// Mitsubishi GX Works2 project: msp_7   PLC: Q03UDV

PROGRAM MAIN
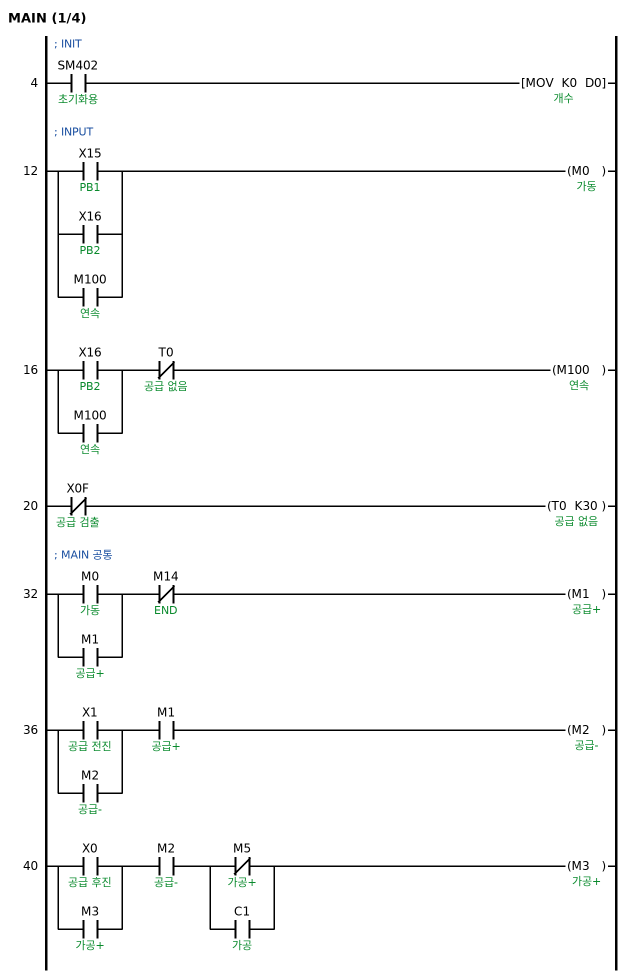
; INIT
4     LD      SM402  ; 초기화용
      MOV     K0 D0  ; 개수
; INPUT
12    LD      X15  ; PB1
      OR      X16  ; PB2
      OR      M100  ; 연속
      OUT     M0  ; 가동
16    LD      X16  ; PB2
      OR      M100  ; 연속
      ANI     T0  ; 공급 없음
      OUT     M100  ; 연속
20    LDI     X0F  ; 공급 검출
      OUT     T0 K30  ; 공급 없음
; MAIN 공통
32    LD      M0  ; 가동
      OR      M1  ; 공급+
      ANI     M14  ; END
      OUT     M1  ; 공급+
36    LD      X1  ; 공급 전진
      OR      M2  ; 공급-
      AND     M1  ; 공급+
      OUT     M2  ; 공급-
40    LD      X0  ; 공급 후진
      OR      M3  ; 가공+
      AND     M2  ; 공급-
      LDI     M5  ; 가공+
      OR      C1  ; 가공
      ANB
      OUT     M3  ; 가공+
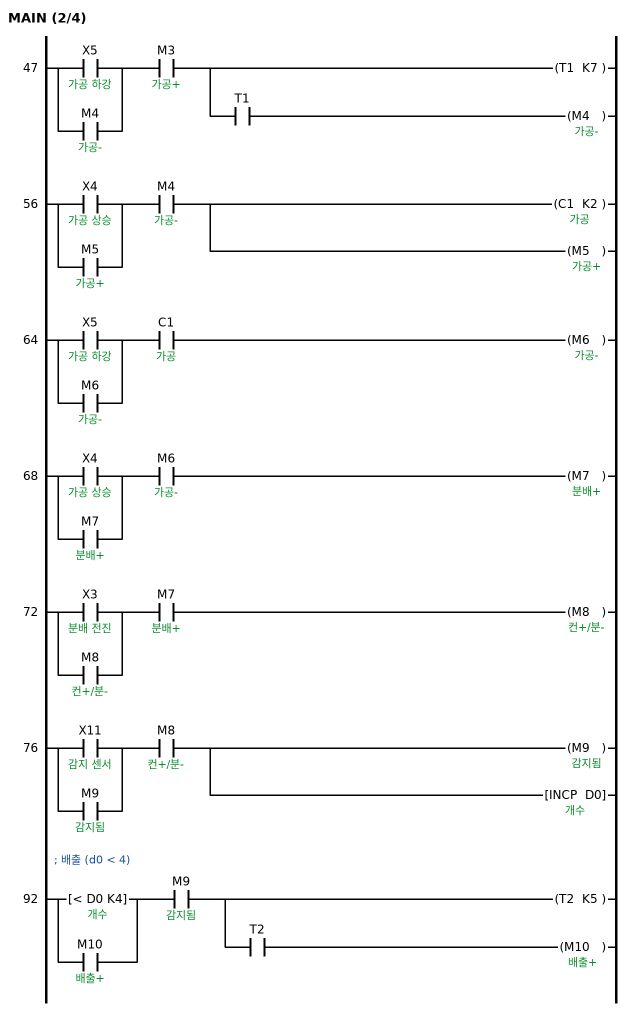
47    LD      X5  ; 가공 하강
      OR      M4  ; 가공-
      AND     M3  ; 가공+
      OUT     T1 K7
      AND     T1
      OUT     M4  ; 가공-
56    LD      X4  ; 가공 상승
      OR      M5  ; 가공+
      AND     M4  ; 가공-
      OUT     C1 K2  ; 가공
      OUT     M5  ; 가공+
64    LD      X5  ; 가공 하강
      OR      M6  ; 가공-
      AND     C1  ; 가공
      OUT     M6  ; 가공-
68    LD      X4  ; 가공 상승
      OR      M7  ; 분배+
      AND     M6  ; 가공-
      OUT     M7  ; 분배+
72    LD      X3  ; 분배 전진
      OR      M8  ; 컨+/분-
      AND     M7  ; 분배+
      OUT     M8  ; 컨+/분-
76    LD      X11  ; 감지 센서
      OR      M9  ; 감지됨
      AND     M8  ; 컨+/분-
      OUT     M9  ; 감지됨
      INCP    D0
; 배출 (d0 < 4)
92    LD<     D0 K4  ; 개수
      OR      M10  ; 배출+
      AND     M9  ; 감지됨
      OUT     T2 K5
      AND     T2
      OUT     M10  ; 배출+
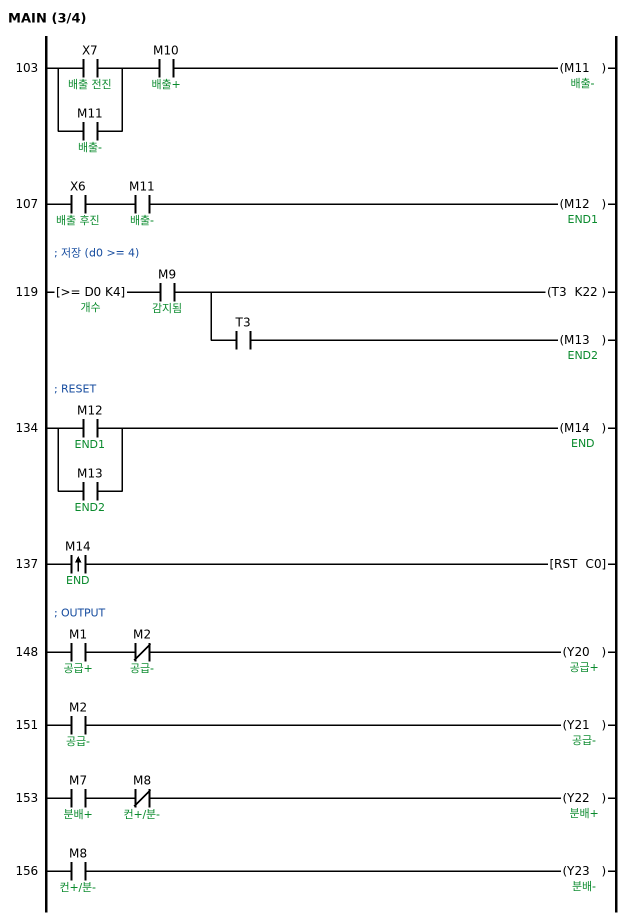
103   LD      X7  ; 배출 전진
      OR      M11  ; 배출-
      AND     M10  ; 배출+
      OUT     M11  ; 배출-
107   LD      X6  ; 배출 후진
      AND     M11  ; 배출-
      OUT     M12  ; END1
; 저장 (d0 >= 4)
119   LD>=    D0 K4  ; 개수
      AND     M9  ; 감지됨
      OUT     T3 K22
      AND     T3
      OUT     M13  ; END2
; RESET
134   LD      M12  ; END1
      OR      M13  ; END2
      OUT     M14  ; END
137   LDP     M14  ; END
      RST     C0
; OUTPUT
148   LD      M1  ; 공급+
      ANI     M2  ; 공급-
      OUT     Y20  ; 공급+
151   LD      M2  ; 공급-
      OUT     Y21  ; 공급-
153   LD      M7  ; 분배+
      ANI     M8  ; 컨+/분-
      OUT     Y22  ; 분배+
156   LD      M8  ; 컨+/분-
      OUT     Y23  ; 분배-
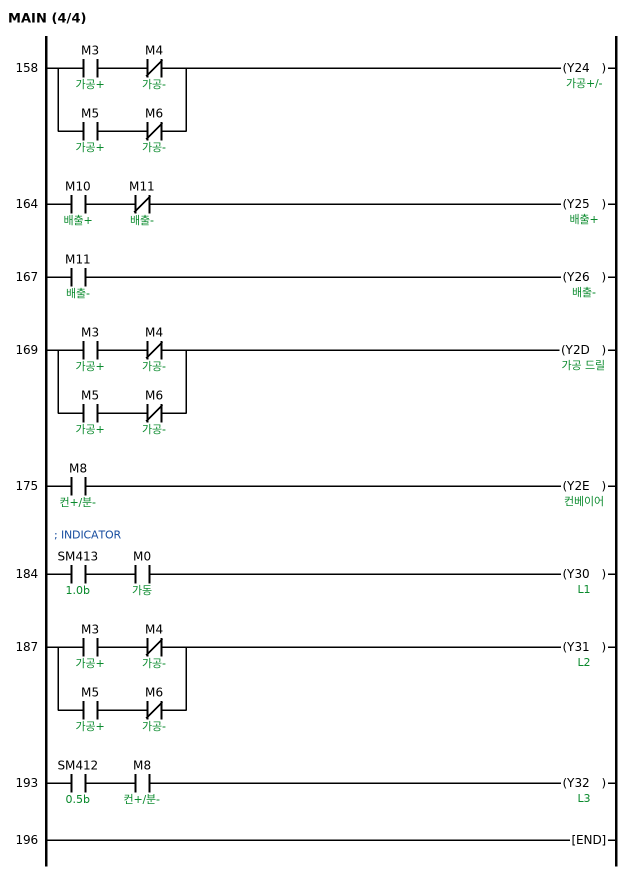
158   LD      M3  ; 가공+
      ANI     M4  ; 가공-
      LD      M5  ; 가공+
      ANI     M6  ; 가공-
      ORB
      OUT     Y24  ; 가공+/-
164   LD      M10  ; 배출+
      ANI     M11  ; 배출-
      OUT     Y25  ; 배출+
167   LD      M11  ; 배출-
      OUT     Y26  ; 배출-
169   LD      M3  ; 가공+
      ANI     M4  ; 가공-
      LD      M5  ; 가공+
      ANI     M6  ; 가공-
      ORB
      OUT     Y2D  ; 가공 드릴
175   LD      M8  ; 컨+/분-
      OUT     Y2E  ; 컨베이어
; INDICATOR
184   LD      SM413  ; 1.0b
      AND     M0  ; 가동
      OUT     Y30  ; L1
187   LD      M3  ; 가공+
      ANI     M4  ; 가공-
      LD      M5  ; 가공+
      ANI     M6  ; 가공-
      ORB
      OUT     Y31  ; L2
193   LD      SM412  ; 0.5b
      AND     M8  ; 컨+/분-
      OUT     Y32  ; L3
196   END
END_PROGRAM

// device comments not shown above
X2  ; 분배 후진
X12  ; 금속 센서
X17  ; PB3
X18  ; PB4
X19  ; PB5
X1A  ; PB6
X1B  ; PB7
X1C  ; PB8
Y27  ; 스톱+/-
Y33  ; L4
Y34  ; L5
Y35  ; L6
Y36  ; L7
Y37  ; BUZZER
C2  ; 마감 가공
D1  ; 금속
